// TIA Portal V16 export
// export: Created 2021-07-12T14:47:19.0053046Z, ExportSetting WithDefaults, DisplayName Totally Integrated Automation Portal, DisplayVersion V16, DisplayName TIA Portal Version Control Interface, DisplayVersion V16, DisplayName TIA Portal Openness, DisplayVersion V16, DisplayName STEP 7 Professional, DisplayVersion V16, DisplayName STEP 7 Safety, DisplayVersion V16, DisplayName WinCC Professional, DisplayVersion V16
TYPE "LSimaHydTO_typePositionControl"
TITLE = LSimaHydTO_typePositionControl
// Position control configuration data
// stored: IsFailsafeCompliant false
   STRUCT
      SmoothingTimeByChangeDifference { S7_SetPoint := 'True'} : LReal;   // Time constant for smoothing manipulated variable jumps [s]
      PreControl { S7_SetPoint := 'True'} : LReal := 100.0;   // Weighting factor of the precontrol Kpc [%]
      ProportionalGain { S7_SetPoint := 'True'} : LReal := 10.0;   // Proportional gain Kp [1/s]
      IntegralTime { S7_SetPoint := 'True'} : LReal;   // Active integral action time Ti [s]
      DerivativeTime { S7_SetPoint := 'True'} : LReal;   // Active derivative action time Td [s]
      DecayTime { S7_SetPoint := 'True'} : LReal := 0.0;   // Decay time constant of the DT1 component [s]
      OutputUppLimit { S7_SetPoint := 'True'} : LReal := 10000.0;   // Manipulated value high limit [unit/s]
      OutputLowLimit { S7_SetPoint := 'True'} : LReal := -10000.0;   // Manipulated value low limit [unit/s]
   END_STRUCT;
END_TYPE
